INTERFACE I_MessageLogger

METHOD LogMessage : String
VAR_INPUT
	Message			: STRING;
END_VAR
END_METHOD

PROPERTY message : string
GET
END_GET
END_PROPERTY

END_INTERFACE

(* stored: Version 1.1.0.1, ProductVersion 3.1.4024.11
   Itf I_MessageLogger: Id {ec655abd-4dec-479e-9b35-4f62bb6f0459}
   Method LogMessage: Id {b07d4e27-c2ca-4837-babc-69109c0637cb}
   Property message: Id {62ddc68c-11f8-4fec-ac9c-2f79cddc580d}
   Get Get: Id {e1ead310-d158-43e2-8941-2df41c16e013} *)
